// TIA Portal V18 export
DATA_BLOCK "HeatingPLC_vAO_Vars"   // DB11002
{ S7_Optimized_Access := 'FALSE' }
VERSION : 0.1
// stored: AutoNumber false, DBAccessibleFromOPCUA true, IsOnlyStoredInLoadMemory false, IsWriteProtectedInAS false
   VAR
      vAO1 { S7_SetPoint := 'True'} : "UDT_vAO";
      vAO2 { S7_SetPoint := 'True'} : "UDT_vAO";
      vAO3 { S7_SetPoint := 'True'} : "UDT_vAO";
      vAO4 { S7_SetPoint := 'True'} : "UDT_vAO";
      vAO5 { S7_SetPoint := 'True'} : "UDT_vAO";
      vAO6 { S7_SetPoint := 'True'} : "UDT_vAO";
      vAO7 { S7_SetPoint := 'True'} : "UDT_vAO";
      vAO8 { S7_SetPoint := 'True'} : "UDT_vAO";
   END_VAR
BEGIN
END_DATA_BLOCK
